FUNCTION_BLOCK Test_TStreamAdd_Read_DINT EXTENDS TUnitTestBase
VAR
    Stream : TStream(StreamLength := 2);
END_VAR



Stream.Init(2);

Stream.Add_DINT(12345678);
    
Assertion.AssertEquals_UDINT(
    Expected := 4,
    Actual := Stream.Position,
    VariableName := 'Stream.Position');
    
Stream.Seek(0);

Assertion.AssertEquals_DINT(
    Expected := 12345678,
    Actual := Stream.Read_DINT(),
    VariableName := 'Stream.Read_DINT()');
    
Assertion.AssertEquals_UDINT(
    Expected := 4,
    Actual := Stream.Position,
    VariableName := 'Stream.Position');
    
    
TestFinished();

END_FUNCTION_BLOCK

(* stored: Version 1.1.0.1, ProductVersion 3.1.4024.4
   POU Test_TStreamAdd_Read_DINT: Id {d17e252a-9da5-4528-a32e-a1282cb1a6bb}, SpecialFunc None *)
